// Mitsubishi GX Works2 project: Ex02   PLC: Q02/Q02H

PROGRAM MAIN
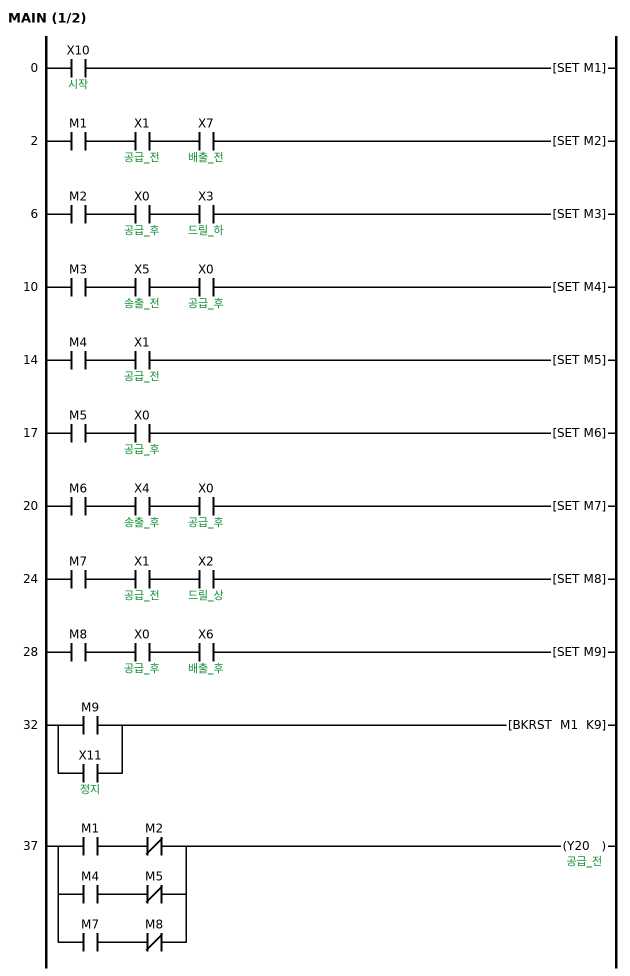
0     LD      X10  ; 시작
      SET     M1
2     LD      M1
      AND     X1  ; 공급_전
      AND     X7  ; 배출_전
      SET     M2
6     LD      M2
      AND     X0  ; 공급_후
      AND     X3  ; 드릴_하
      SET     M3
10    LD      M3
      AND     X5  ; 송출_전
      AND     X0  ; 공급_후
      SET     M4
14    LD      M4
      AND     X1  ; 공급_전
      SET     M5
17    LD      M5
      AND     X0  ; 공급_후
      SET     M6
20    LD      M6
      AND     X4  ; 송출_후
      AND     X0  ; 공급_후
      SET     M7
24    LD      M7
      AND     X1  ; 공급_전
      AND     X2  ; 드릴_상
      SET     M8
28    LD      M8
      AND     X0  ; 공급_후
      AND     X6  ; 배출_후
      SET     M9
32    LD      M9
      OR      X11  ; 정지
      BKRST   M1 K9
37    LD      M1
      ANI     M2
      LD      M4
      ANI     M5
      ORB
      LD      M7
      ANI     M8
      ORB
      OUT     Y20  ; 공급_전
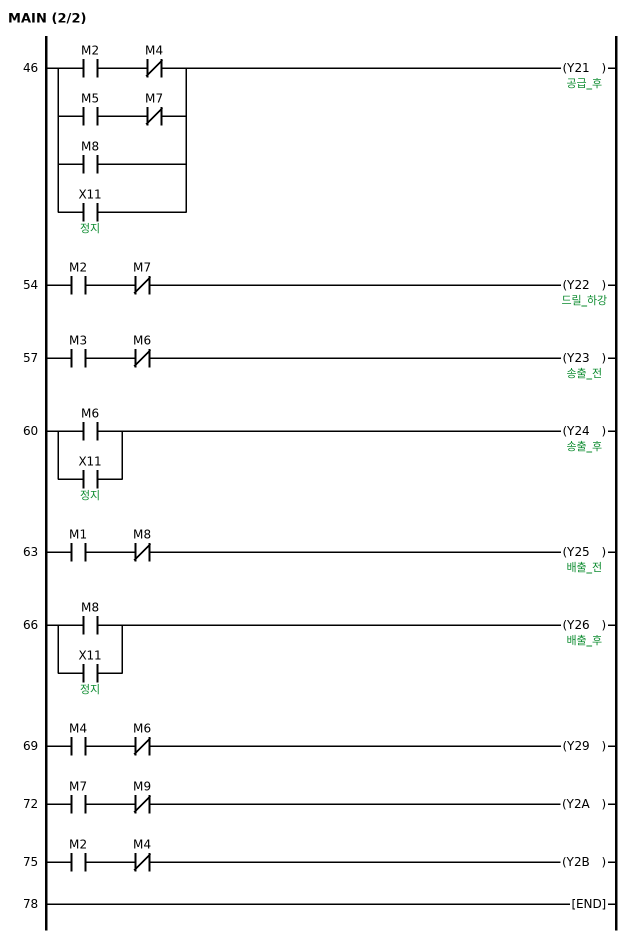
46    LD      M2
      ANI     M4
      LD      M5
      ANI     M7
      ORB
      OR      M8
      OR      X11  ; 정지
      OUT     Y21  ; 공급_후
54    LD      M2
      ANI     M7
      OUT     Y22  ; 드릴_하강
57    LD      M3
      ANI     M6
      OUT     Y23  ; 송출_전
60    LD      M6
      OR      X11  ; 정지
      OUT     Y24  ; 송출_후
63    LD      M1
      ANI     M8
      OUT     Y25  ; 배출_전
66    LD      M8
      OR      X11  ; 정지
      OUT     Y26  ; 배출_후
69    LD      M4
      ANI     M6
      OUT     Y29
72    LD      M7
      ANI     M9
      OUT     Y2A
75    LD      M2
      ANI     M4
      OUT     Y2B
78    END
END_PROGRAM
